// TIA Portal V18 export
FUNCTION "analogScale" : Void   // FC1, LAD
{ S7_Optimized_Access := 'TRUE' }
// stored: SetENOAutomatically false
   VAR_INPUT
      minSensor : Real;
      maxSensor : Real;
      rawValue : Int;
   END_VAR
   VAR_OUTPUT
      scaledValue : Real;
   END_VAR
   VAR_TEMP
      tempNormalizedValue : Real;
   END_VAR
BEGIN

REGION Network 1
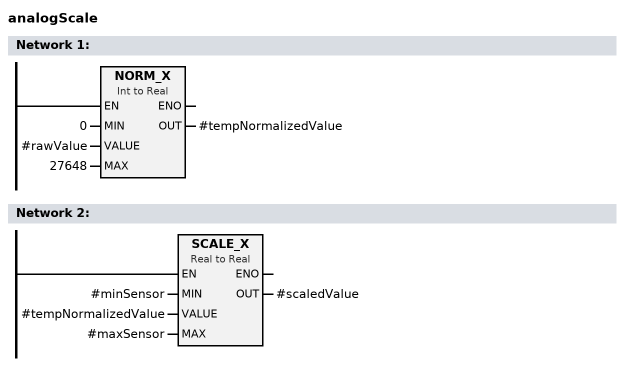
   RUNG wire#powerrail
      { S7_Templates := "[SrcType := Int, DestType := Real]" } Normalize(min := 0, value := #rawValue, max := 27648, out => #tempNormalizedValue)
   END_RUNG
   // the same network as SCL:
   #tempNormalizedValue := NORM_X(MIN := 0, VALUE := #rawValue, MAX := 27648);
END_REGION

REGION Network 2
   RUNG wire#powerrail
      { S7_Templates := "[SrcType := Real, DestType := Real]" } Scale(min := #minSensor, value := #tempNormalizedValue, max := #maxSensor, out => #scaledValue)
   END_RUNG
   // the same network as SCL:
   #scaledValue := SCALE_X(MIN := #minSensor, VALUE := #tempNormalizedValue, MAX := #maxSensor);
END_REGION
END_FUNCTION
